Fanuc KAREL source: kt00122.compact.KL

PROGRAM KT00122
%STACKSIZE=65535
%PRIORITY=65535
%NOLOCKGROUP
VAR
H1 : ARRAY[2] OF SHORT
I2 : INTEGER
OUT : REAL
BEGIN
H1[1]=2
I2=3
OUT=((H1[1]) / (I2))
END KT00122
